METHOD PUBLIC PreExecutionCheck
VAR_INPUT
	Check : I_PreExecutionChecks;
END_VAR
Check.IsTrue(ipSrcImage.IsValid, 'ipSrcImage must contain an image');
END_METHOD

END_FUNCTION_BLOCK

// Nodes/Image Segmentation/Node_F_VN_Threshold
{attribute 'linkalways'} 
{attribute 'no_explicit_call' := 'This FB is a CLASS and must be accessed using methods or properties'}
{attribute 'enable_dynamic_creation'}
FUNCTION_BLOCK Node_F_VN_Threshold EXTENDS VisionNode
VAR
	ipSrcImage : _ITcVnImage;
    ipDestImage : _ITcVnImage;
    fThreshold : _LREAL(0.0);
    fMaxValue : _LREAL(0.0);
	eThresholdType : _ETcVnThresholdType(ETcVnThresholdType.TCVN_TT_BINARY);
    hrPrev : _HRESULT(S_OK);
	hresult : _HRESULT(S_OK);
END_VAR

METHOD FB_init : BOOL
VAR_INPUT
	bInitRetains : BOOL; // if TRUE, the retain variables are initialized (warm start / cold start)
	bInCopyCode : BOOL;  // if TRUE, the instance afterwards gets moved into the copy code (online change)
END_VAR
AddInput('ipSrcImage', ipSrcImage);
AddInput('hrPrev', hrPrev);
AddParameter('fThreshold', fThreshold);
AddParameter('fMaxValue', fMaxValue);
AddParameter('eThresholdType', eThresholdType);
AddOutput('ipDestImage', ipDestImage);
AddOutput('hresult',hresult);
END_METHOD

METHOD PUBLIC  Clone : I_Node
VAR
	pNode : POINTER TO Node_F_VN_Threshold;
END_VAR
pNode := __NEW(Node_F_VN_Threshold);
Clone := pNode^;
END_METHOD

METHOD PROTECTED  OnExecute : HRESULT
hresult.Value := F_VN_Threshold(
	ipSrcImage := ipSrcImage.Value, 
	ipDestImage := ipDestImage.Value, 
	fThreshold := fThreshold.Value, 
	fMaxValue := fMaxValue.Value, 
	eThresholdType := eThresholdType.Value, 
	hrPrev:= hrPrev.Value);
END_METHOD

METHOD PUBLIC PreExecutionCheck
VAR_INPUT
	Check : I_PreExecutionChecks;
END_VAR
Check.IsTrue(ipSrcImage.IsValid, 'ipSrcImage must contain an image');
//Check.IsTrue(ipSrcImage.IsPixelValueCompatible(fThreshold.Value), 'The value of fThreshold is not compatible with the source image pixel depth');
//Check.IsTrue(ipSrcImage.IsPixelValueCompatible(fMaxValue.Value), 'The value of fMaxValue is not compatible with the source image pixel depth');
END_METHOD

END_FUNCTION_BLOCK

// Nodes/VisionNodePack
{attribute 'linkalways'} 
{attribute 'no_explicit_call' := 'This FB is a CLASS and must be accessed using methods or properties'}
{attribute 'enable_dynamic_creation'}
FUNCTION_BLOCK VisionNodePack IMPLEMENTS I_NodePack
VAR
    // Algebraic Container Operations
    
    // Algebraic Image Operations
    node_F_VN_BitwiseNotImage : Node_F_VN_BitwiseNotImage;
        
    // Basic Container Operations
    node_F_VN_AppendToContainer_DINT : Node_F_VN_AppendToContainer_DINT;
    node_F_VN_AppendToContainer_INT : Node_F_VN_AppendToContainer_INT;
    
    // Basic Image Operations
    node_F_VN_CopyImage : Node_F_VN_CopyImage;
    node_F_VN_GetImageChannel : Node_F_VN_GetImageChannel;
    node_F_VN_GetImageHeight : Node_F_VN_GetImageHeight;
    node_F_VN_GetImageInfo : Node_F_VN_GetImageInfo;
    node_F_VN_GetImageWidth : Node_F_VN_GetImageWidth;
    
    // Code Quality
    
    // Code Reading
    // node_F_VN_ReadBarcode : Node_F_VN_ReadBarcode
    // node_F_VN_ReadBarcodeExp : Node_F_VN_ReadBarcodeExp
    // node_F_VN_ReadBarcodeExp2 : Node_F_VN_ReadBarcodeExp2
    // node_F_VN_ReadDataMatrixCode : Node_F_VN_ReadDataMatrixCode
    // node_F_VN_ReadDataMatrixCodeExp : Node_F_VN_ReadDataMatrixCodeExp
    // node_F_VN_ReadDataMatrixCodeExp2 : Node_F_VN_ReadDataMatrixCodeExp2
    // node_F_VN_ReadPharmaCode : Node_F_VN_ReadPharmaCode
    // node_F_VN_ReadPharmaCodeExp : Node_F_VN_ReadPharmaCodeExp
    // node_F_VN_ReadPharmaCodeExp2 : Node_F_VN_ReadPharmaCodeExp2
    // node_F_VN_ReadQRCode : Node_F_VN_ReadQRCode
    // node_F_VN_ReadQRCodeExp : Node_F_VN_ReadQRCodeExp
    // node_F_VN_ReadQRCodeExp2 : Node_F_VN_ReadQRCodeExp2
    
    // Container Statistics
    
    // Contour Analysis
    
    // Control Functions
    
    // Drawing
    node_F_VN_DrawContours : Node_F_VN_DrawContours;
    node_F_VN_DrawLine : Node_F_VN_DrawLine;
    node_F_VN_PutLabel : Node_F_VN_PutLabel;
    node_F_VN_PutText : Node_F_VN_PutText;
    
    // Fourier Analysis
    
    // Geometric and Coordinate Transformations
    node_F_VN_FlipImage : Node_F_VN_FlipImage;
    
    // Image Analysis
    node_F_VN_DetectBlobs : Node_F_VN_DetectBlobs;
    
    // Image Color and Contrast Processing
    node_F_VN_ConvertColorSpace : Node_F_VN_ConvertColorSpace;
    node_F_VN_ApplyColorMap : Node_F_VN_ApplyColorMap;
    node_F_VN_GenerateColorMap : Node_F_VN_GenerateColorMap;
    
    // Image Filtering
    node_F_VN_BoxFilter : Node_F_VN_BoxFilter;
    node_F_VN_GaussianFilter : Node_F_VN_GaussianFilter;
    node_F_VN_LaplacianFilter : Node_F_VN_LaplacianFilter;
    
    // Image Segmentation
    node_F_VN_Threshold : Node_F_VN_Threshold;
    
    // Keypoint Features
    
    // Machine Learning
    
    // Measurement
    
    // Miscellaneous
    
    // OCR
    
    // Texture Analysis
 
END_VAR

METHOD PUBLIC RegisterWithNodeFactory
VAR_INPUT
	NodeFactory : I_NodeFactory;
END_VAR
// Algebraic Container Operations

// Algebraic Image Operations
NodeFactory.AddNodeAsPrototype('Vision/Algebraic Image Operations/F_VN_BitwiseNotImage', node_F_VN_BitwiseNotImage);

// Basic Container Operations
NodeFactory.AddNodeAsPrototype('Vision/Basic Container Operations/F_VN_AppendToContainer/F_VN_AppendToContainer_DINT', node_F_VN_AppendToContainer_DINT);
NodeFactory.AddNodeAsPrototype('Vision/Basic Container Operations/F_VN_AppendToContainer/F_VN_AppendToContainer_INT', node_F_VN_AppendToContainer_INT);

// Basic Image Operations
NodeFactory.AddNodeAsPrototype('Vision/Basic Image Operations/F_VN_CopyImage', node_F_VN_CopyImage);
NodeFactory.AddNodeAsPrototype('Vision/Basic Image Operations/F_VN_GetImageChannel', node_F_VN_GetImageChannel);
NodeFactory.AddNodeAsPrototype('Vision/Basic Image Operations/F_VN_GetImageHeight', node_F_VN_GetImageHeight);
NodeFactory.AddNodeAsPrototype('Vision/Basic Image Operations/F_VN_GetImageInfo', node_F_VN_GetImageInfo);
NodeFactory.AddNodeAsPrototype('Vision/Basic Image Operations/F_VN_GetImageWidth', node_F_VN_GetImageWidth);
 
// Code Quality

// Code Reading

// Container Statistics

// Contour Analysis

// Control Functions
    
// Drawing
NodeFactory.AddNodeAsPrototype('Vision/Drawing/F_VN_DrawContours', node_F_VN_DrawContours);
NodeFactory.AddNodeAsPrototype('Vision/Drawing/F_VN_DrawLine', node_F_VN_DrawLine);
NodeFactory.AddNodeAsPrototype('Vision/Drawing/F_VN_PutLabel', node_F_VN_PutLabel);
NodeFactory.AddNodeAsPrototype('Vision/Drawing/F_VN_PutText', node_F_VN_PutText);

// Fourier Analysis

// Geometric and Coordinate Transformations
NodeFactory.AddNodeAsPrototype('Vision/Geometric and Coordinate Transformations/F_VN_FlipImage', node_F_VN_FlipImage);

// Image Analysis
NodeFactory.AddNodeAsPrototype('Vision/Image Analysis/Object Detection/F_VN_DetectBlobs', node_F_VN_DetectBlobs);

// Image Color and Contrast Processing
NodeFactory.AddNodeAsPrototype('Vision/Image Color and Contrast Processing/F_VN_ConvertColorSpace', node_F_VN_ConvertColorSpace);
NodeFactory.AddNodeAsPrototype('Vision/Image Color and Contrast Processing/F_VN_ApplyColorMap', node_F_VN_ApplyColorMap);
NodeFactory.AddNodeAsPrototype('Vision/Image Color and Contrast Processing/F_VN_GenerateColorMap', node_F_VN_GenerateColorMap);

// Image Filtering
NodeFactory.AddNodeAsPrototype('Vision/Image Filtering/F_VN_BoxFilter', node_F_VN_BoxFilter);
NodeFactory.AddNodeAsPrototype('Vision/Image Filtering/F_VN_GaussianFilter', node_F_VN_GaussianFilter);
NodeFactory.AddNodeAsPrototype('Vision/Image Filtering/F_VN_LaplacianFilter', node_F_VN_LaplacianFilter);
    
// Image Segmentation
NodeFactory.AddNodeAsPrototype('Vision/Image Segmentation/F_VN_Threshold', node_F_VN_Threshold);

// Keypoint Features

// Machine Learning

// Measurement

// Miscellaneous

// OCR

// Texture Analysis
END_METHOD

END_FUNCTION_BLOCK

// VisionPack
{attribute 'linkalways'} 
{attribute 'no_explicit_call' := 'This FB is a CLASS and must be accessed using methods or properties'}
{attribute 'enable_dynamic_creation'}
FUNCTION_BLOCK VisionPack IMPLEMENTS I_GraphPack
VAR
	visionDatatypePack : VisionDatatypePack;
	visionNodePack : VisionNodePack;
END_VAR

METHOD RegisterWithDatatypes
VAR_INPUT
	Datatypes : I_Datatypes;
END_VAR
visionDatatypePack.RegisterWithDatatypes(Datatypes);
END_METHOD

METHOD PUBLIC RegisterWithNodeFactory
VAR_INPUT
	NodeFactory : I_NodeFactory;
END_VAR
visionNodePack.RegisterWithNodeFactory(NodeFactory);
END_METHOD

END_FUNCTION_BLOCK
